TYPE Ax_Palletizer_Basic_Parameters :
STRUCT
	Vel 	: REAL;
	Acc 	: REAL;
	Dec 	: REAL;
	Jerk 	: REAL;
	Torque 	: REAL;
END_STRUCT
END_TYPE

(* stored: Version 1.1.0.1, ProductVersion 3.1.4024.11
   DUT Ax_Palletizer_Basic_Parameters: Id {54fad531-b367-401f-87e1-22bd8b2b262c} *)
